// TIA Portal V21 export
DATA_BLOCK "CV15"   // DB209
{ S7_Optimized_Access := 'TRUE' }
// stored: AutoNumber false, MemoryReserve 100
   VAR
      Tag_IB89 : Byte;
      Tag_IB90 : Byte;
      Tag_IB93 : Byte;
      Tag_IB94 : Byte;
      Tag_IB96 : Byte;
      Tag_IB97 : Byte;
      Tag_IB98 : Byte;
      Tag_MD124 : DInt;
      Tag_MD300 : DInt;
      Tag_MD304 : DInt;
      Tag_MD308 : DInt;
      Tag_MD312 : Real;
      Tag_MD316 : Real;
      Tag_MD320 : DInt;
      Tag_MD324 : DInt;
      Tag_MD340 : DInt;
      Tag_MD344 : DInt;
      Tag_MD348 { ExternalWritable := 'False'} : DInt;
      Tag_MD352 : Real;
      Tag_MD356 : Real;
   END_VAR
BEGIN
END_DATA_BLOCK
